# EPICS IOC start-up script: iocsh/ethercatmcEL6688-PTP-twincat-ads.iocsh
dbLoadRecords("ethercatmcEL6688-PTP-twincat-ads.template", "P=$(P), R=$(R), MOTOR_PORT=$(MOTOR_PORT), ASYN_PORT=$(ASYN_PORT)")
